FUNCTION_BLOCK FB_ParameterFileHandler EXTENDS FB_ParameterHandler
VAR CONSTANT
	sCSVFileHeader 	: STRING := 'NUMBER;NAME;TYPE;DESCRIPTION;FACTORY;MAXIMUM;MINIMUM;UNIT;VALUE$L';
	CSV_FIELDS 		: UINT := 9;
END_VAR
VAR_OUTPUT
	// State outputs
	bInitialized 	: BOOL;
	bError			: BOOL;
	sErrorMessage	: STRING;
END_VAR
VAR
	// States
	eState 		: E_ParameterHandlerState := E_ParameterHandlerState.InitializeFBs;
	
	// Commands
	bCmdInit 	: BOOL;
	
	// File function blocks (asynchronous)
	fbFileOpen	: FB_FileOpen; // https://infosys.beckhoff.com/content/1033/tcplclib_tc2_system/30977547.html
	fbFileWrite	: FB_FileWrite; // https://infosys.beckhoff.com/content/1033/tcplclib_tc2_system/30986763.html
	fbFileClose	: FB_FileClose; // https://infosys.beckhoff.com/content/1033/tcplclib_tc2_system/30972939.html
	fbFileGets	: FB_FileGets; // https://infosys.beckhoff.com/content/1033/tcplclib_tc2_system/30976011.html

	// CSV handling function blocks
	fbCsvMemBufReader : FB_CSVMemBufferReader; // https://infosys.beckhoff.com/content/1033/tcplclib_tc2_utilities/34977931.html
	fbCsvMemBufWriter : FB_CSVMemBufferWriter; // https://infosys.beckhoff.com/content/1033/tcplclib_tc2_utilities/34979467.html

	// Miscelleanous
	nIdxPar  : UINT; // Parameter array iterator
	sCsvRecord : T_MaxString := ''; // String buffer (single CSV text line)
	bHeaderRead : BOOL; // TRUE once the CSV header line has been read
END_VAR

ExecStateMachine();

METHOD PRIVATE ExecStateMachine : BOOL
VAR
	i 					: UINT; // Iterator
	pParameter 			: POINTER TO Udt_Parameter; // Temporary pointer to parameter
	sParameterFromFile 	: Udt_Parameter; // Parameter retrieved from file
	sCSVField 			: T_MaxString; // Single CSV field value (record field)
	bMatch 				: BOOL;
END_VAR
// Parameter file handler state machine
CASE eState OF
	E_ParameterHandlerState.InitializeFBs:
		// Initialize function blocks
		fbFileOpen(
			bExecute := FALSE,
			ePath := PATH_GENERIC,
		);
		fbFileWrite(
			bExecute := FALSE,
			pWriteBuff := ADR(sCsvRecord)
		);
		fbFileClose(bExecute := FALSE);
		fbFileGets(bExecute := FALSE);

		fbCsvMemBufWriter.pBuffer := ADR(sCsvRecord);
		fbCsvMemBufReader.pBuffer := ADR(sCsvRecord);
		fbCsvMemBufWriter.cbBuffer := SIZEOF(sCsvRecord) - 1;
		fbCsvMemBufReader.cbBuffer := SIZEOF(sCsvRecord);
	
		eState := E_ParameterHandlerState.WaitForCommand;

	E_ParameterHandlerState.WaitForCommand:
		IF bCmdInit THEN
			eState := E_ParameterHandlerState.OpenExistingFile;
		END_IF	

	E_ParameterHandlerState.OpenExistingFile:
		fbFileOpen(
			bExecute := TRUE,	
			sPathName := GVL_Parameters.sPARLIST_FILE,
			nMode := FOPEN_MODEREAD OR FOPEN_MODETEXT, // Open file in read only text mode
		);

		IF (NOT fbFileOpen.bBusy) THEN
			fbFileOpen(bExecute := FALSE);

			IF fbFileOpen.bError THEN
				// Check error codes
				IF (fbFileOpen.nErrId = 16#70C) THEN
					// File not found
					eState := E_ParameterHandlerState.CreateFile;
				ELSE
					sErrorMessage := 'Unable to open file';
					eState := E_ParameterHandlerState.Error;
				END_IF
			ELSE
				nIdxPar := 0;
				bHeaderRead := FALSE;
				eState := E_ParameterHandlerState.ReadRecord;
			END_IF
		END_IF

	E_ParameterHandlerState.CreateFile:
		fbFileOpen(
			bExecute := TRUE,	
			sPathName := GVL_Parameters.sPARLIST_FILE,
			nMode := FOPEN_MODEWRITE OR FOPEN_MODETEXT, // Open file in read/write text mode
		);

		IF (NOT fbFileOpen.bBusy) THEN
			fbFileOpen(bExecute := FALSE);

			IF fbFileOpen.bError THEN
				sErrorMessage := 'Unable to create file';
				eState := E_ParameterHandlerState.Error;
			ELSE		
				fbFileWrite.hFile := fbFileOpen.hFile;
				nIdxPar := 0;
				eState := E_ParameterHandlerState.WriteRecord;
			END_IF
		END_IF
		
	E_ParameterHandlerState.WriteRecord:
		// Code based on Beckhoff example: https://infosys.beckhoff.com/content/1033/tcplclib_tc2_utilities/34979467.html
		sCsvRecord := '';
		fbCsvMemBufWriter.eCmd := eEnumCmd_First; // Write first field value

		IF (nIdxPar > nNumberOfParameters) THEN
			// Done (all parameters were added)
			eState := E_ParameterHandlerState.CloseFile;
		ELSIF (nIdxPar = 0) THEN
			// First line: write the CSV header
			sCsvRecord := sCSVFileHeader;
			eState := E_ParameterHandlerState.WriteRecordBusy;
		ELSE
			// Add the next parameter
			pParameter := arParameters[nIdxPar].pParameter;
			IF (pParameter = 0) THEN
				sErrorMessage := 'Unexpected null pointer';
				eState := E_ParameterHandlerState.Error;
			ELSE
				// We're good to go, iterate over all record fields
				FOR i := 1 TO CSV_FIELDS DO 
					CASE i OF
						1: sCSVField := UDINT_TO_STRING(pParameter^.nNumber);
						2: sCSVField := pParameter^.sName;
						3: sCSVField := pParameter^.sType;
						4: sCSVField := pParameter^.sDiscription;
						5: sCSVField := LREAL_TO_STRING(pParameter^.fFactory);
						6: sCSVField := LREAL_TO_STRING(pParameter^.fMaximum);
						7: sCSVField := LREAL_TO_STRING(pParameter^.fMinimum);
						8: sCSVField := pParameter^.sUnit;
						9: sCSVField := LREAL_TO_STRING(pParameter^.fValue);
					END_CASE
					sCSVField := STRING_TO_CSVFIELD(sCSVField, FALSE);
					
					// Add new field to the record buffer
					fbCsvMemBufWriter(
						putValue := sCSVField,
						bCRLF := (i = CSV_FIELDS) // Write CRLF after the last field value 
					);
					IF fbCsvMemBufWriter.bOk THEN
						fbCsvMemBufWriter.eCmd := eEnumCmd_Next;
					ELSE // Error
						sErrorMessage := 'Unable to store fields in CSV buffer';
						eState := E_ParameterHandlerState.Error;
						RETURN;
					END_IF
	
				END_FOR

				eState := E_ParameterHandlerState.WriteRecordBusy;
			END_IF;
		END_IF;

	E_ParameterHandlerState.WriteRecordBusy:
		fbFileWrite(bExecute := TRUE, cbWriteLen := INT_TO_UDINT(LEN(sCsvRecord)));
		IF (NOT fbFileWrite.bBusy) THEN
			fbFileWrite(bExecute := FALSE);
			IF fbFileWrite.bError THEN
				sErrorMessage := 'Unable to write record to file';
				eState := E_ParameterHandlerState.Error;
			ELSE		
				nIdxPar := nIdxPar + 1;	 
				eState := E_ParameterHandlerState.WriteRecord;
			END_IF
		END_IF
		
	E_ParameterHandlerState.ReadRecord:
		fbFileGets(bExecute := TRUE, hFile := fbFileOpen.hFile);
		IF (NOT fbFileGets.bBusy) THEN
			sCsvRecord := fbFileGets.sLine;
			fbFileGets(bExecute := FALSE);
			IF fbFileGets.bError THEN
				sErrorMessage := 'Unable to read line from file';
				eState := E_ParameterHandlerState.Error;
			ELSIF fbFileGets.bEOF THEN
				// Finished reading the file
				eState := E_ParameterHandlerState.CloseFile;			
			ELSIF NOT bHeaderRead THEN 
				// Skip first line (header)
				bHeaderRead := TRUE;
			ELSE
				eState := E_ParameterHandlerState.ParseRecord;
			END_IF
		END_IF

	E_ParameterHandlerState.ParseRecord:
		fbCsvMemBufReader.eCmd := eEnumCmd_First; // Read first field value

		FOR i := 1 TO CSV_FIELDS DO 
			// Read field from the record buffer
			fbCsvMemBufReader(getValue => sCSVField);
			IF fbCsvMemBufReader.bOk THEN
				sCSVField := CSVFIELD_TO_STRING(sCSVField, FALSE);
				CASE i OF
					1: sParameterFromFile.nNumber := STRING_TO_UDINT(sCSVField);
					2: sParameterFromFile.sName := sCSVField;
					3: sParameterFromFile.sType := sCSVField;
					4: sParameterFromFile.sDiscription := sCSVField;
					5: sParameterFromFile.fFactory := STRING_TO_LREAL(sCSVField);
					6: sParameterFromFile.fMaximum := STRING_TO_LREAL(sCSVField);
					7: sParameterFromFile.fMinimum := STRING_TO_LREAL(sCSVField);
					8: sParameterFromFile.sUnit := sCSVField;
					9: sParameterFromFile.fValue := STRING_TO_LREAL(sCSVField);
				END_CASE
				
				fbCsvMemBufReader.eCmd := eEnumCmd_Next;
			ELSE // Error
				sErrorMessage := 'Unable to parse all CSV fields';
				eState := E_ParameterHandlerState.Error;
				RETURN;
			END_IF
		END_FOR
			
		// Done reading parameter from file. Search for parameter in the PLC parameter array, and copy values.
		FOR i := 1 TO nNumberOfParameters DO
			pParameter := arParameters[i].pParameter;
			IF (pParameter = 0) THEN
				// Unexpected null pointer
				EXIT;
			ELSIF (sParameterFromFile.nNumber = pParameter^.nNumber) THEN
				bMatch := TRUE;
				pParameter^.sName := sParameterFromFile.sName;
				pParameter^.sType := sParameterFromFile.sType;
				pParameter^.sDiscription := sParameterFromFile.sDiscription;
				pParameter^.fFactory := sParameterFromFile.fFactory;
				pParameter^.fMaximum := sParameterFromFile.fMaximum;
				pParameter^.fMinimum := sParameterFromFile.fMinimum;
				pParameter^.sUnit := sParameterFromFile.sUnit;
				pParameter^.fValue := sParameterFromFile.fValue;
				EXIT;
			END_IF
		END_FOR

		IF bMatch THEN
			// Finished, move to the next record		
			eState := E_ParameterHandlerState.ReadRecord;
		ELSE
			sErrorMessage := 'Parameter in CSV file not found in PLC';
			eState := E_ParameterHandlerState.Error;
		END_IF
	
	E_ParameterHandlerState.CloseFile:
		fbFileClose(bExecute := TRUE, hFile := fbFileOpen.hFile);
		IF (NOT fbFileClose.bBusy) THEN
			fbFileClose(bExecute := FALSE);
			IF fbFileClose.bError THEN
				sErrorMessage := 'Unable to close file'; 
				eState := E_ParameterHandlerState.Error;
			ELSE
				bInitialized S= bCmdInit;
				eState := E_ParameterHandlerState.WaitForCommand;
			END_IF
		END_IF
	
	E_ParameterHandlerState.Error:
		IF (sErrorMessage = '') THEN
			sErrorMessage := 'Unknown error';
		END_IF
		;
END_CASE

bError := (eState = E_ParameterHandlerState.Error);
END_METHOD

METHOD PUBLIC Init : BOOL
bCmdInit := NOT bInitialized;
Init := bInitialized;
END_METHOD

END_FUNCTION_BLOCK

(* stored: Version 1.1.0.1, ProductVersion 3.1.4024.11
   POU FB_ParameterFileHandler: Id {052dee22-c06d-0a14-2ec0-25219a011600}, SpecialFunc None
   Folder Commands: Id {bcbefad3-29cb-0730-1187-e3aea827e983}
   Folder Private: Id {11dd7ad9-4d84-0833-08cb-6ecb397bdce4}
   Method ExecStateMachine: Id {56cdb778-6ecd-014e-21b9-022e7b6f4d2c}
   Method Init: Id {d9fae5f4-5172-06d7-1319-23a49bf2ac18} *)
